FUNCTION_BLOCK FB_MotorSimple EXTENDS FB_Base
VAR_INPUT
END_VAR
VAR_OUTPUT
END_VAR
VAR
END_VAR

//FB_Init ist immer implizit verfügbar und wird primär für die Initialisierung verwendet.
//Der Rückgabewert wird nicht ausgewertet. Für gezielte Einflussnahme können Sie
//die Methoden explizit deklarieren und darin mit dem Standard-Initialisierungscode 
//zusätzlichen Code bereitstellen. Sie können den Rückgabewert auswerten.
METHOD FB_Init: BOOL
VAR_INPUT    
	bInitRetains					: BOOL; 					// TRUE: Die Retain-Variablen werden initialisiert (Reset warm / Reset kalt)    
	bInCopyCode						: BOOL;  					// TRUE: Die Instanz wird danach in den Kopiercode kopiert (Online-Change)
	
	I_Name                : STRING;         //  Name
	I_ID                  : UINT;            // ID
END_VAR
END_METHOD

END_FUNCTION_BLOCK

(* stored: Version 1.1.0.1, ProductVersion 3.1.4026.18
   POU FB_MotorSimple: Id {f28d4450-f9e9-4af2-bbaf-1853171416fe}, SpecialFunc None
   Folder 01 Properties: Id {bd17f19f-4bc5-4ff6-ba2e-b001df3129e1}
   Folder 02 Methodes: Id {ff9e3ec7-8f18-43cf-96ff-a8b9f5e98df5}
   Method FB_Init: Id {d47ef4d2-3135-4a9f-954d-3322b239918f} *)
